FUNCTION_BLOCK Elevator
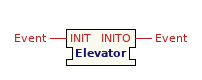
  EVENT_INPUT
    INIT;
  END_EVENT
  EVENT_OUTPUT
    INITO;
  END_EVENT
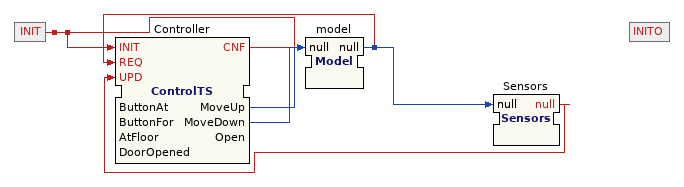
  FBS
    model : Model;
    Controller : ControlTS;
    Sensors : Sensors;
  END_FBS
  EVENT_CONNECTIONS
    INIT TO model.null;
    INIT TO Controller.INIT;
    model.null TO Controller.REQ;
    Controller.CNF TO model.null;
    model.null TO Sensors.null;
    model.null TO Sensors.null;
    Sensors.null TO Controller.UPD;
  END_CONNECTIONS
  DATA_CONNECTIONS
    Controller.MoveUp TO model.null;
    Controller.MoveDown TO model.null;
    model.null TO Sensors.null;
  END_CONNECTIONS
END_FUNCTION_BLOCK
